SYSTEM ASM_MVCDR (* Assembly System Control+Diagnostics+HMI with Remote Model+View *)
  (* Standard: 61499-1; Classification: Simulation; ApplicationDomain: Assembly; Type: Dual Stroke Cylinder *)
  (* Version 0.1, 2004-10-21, JHC, Rockwell Automation, Adapted to new Load/Unload model. *)
  (* Version 0.0, 2004-09-26, JHC, Rockwell Automation, Extended from ASM_MVCDL1. *)
  DEVICE DIAGNOSTICS : FRAME_DEVICE
    RESOURCE IO : EMB_RES
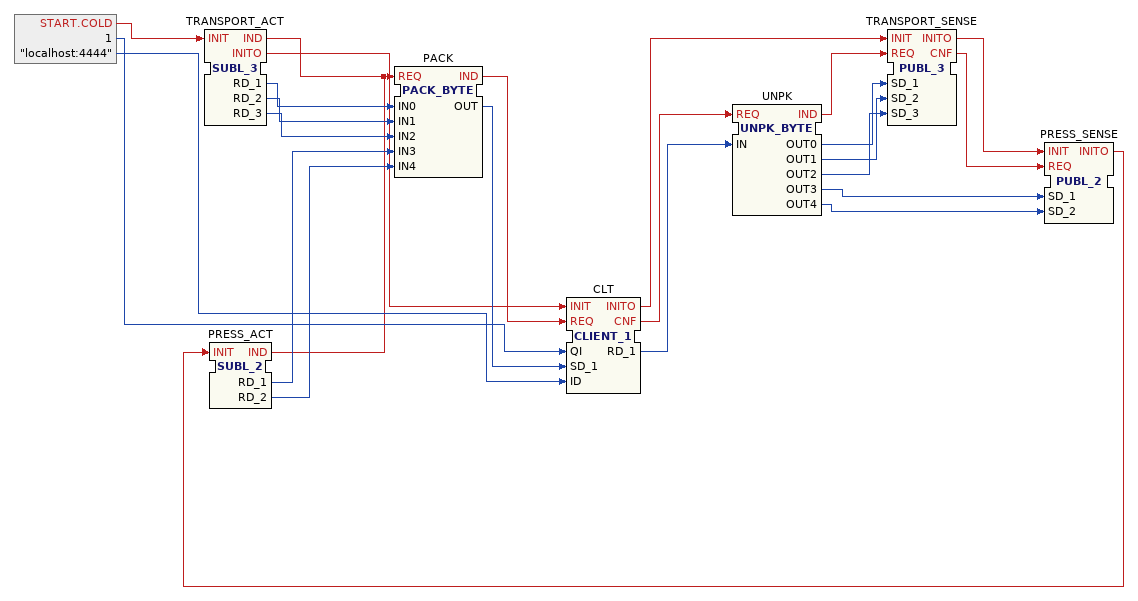
      FBS
        TRANSPORT_SENSE : PUBL_3;
        TRANSPORT_ACT : SUBL_3;
        PRESS_ACT : SUBL_2;
        PRESS_SENSE : PUBL_2;
        PACK : PACK_BYTE;
        CLT : CLIENT_1;
        UNPK : UNPK_BYTE;
      END_FBS
      EVENT_CONNECTIONS
        START.COLD TO TRANSPORT_ACT.INIT;
        TRANSPORT_ACT.IND TO PACK.REQ;
        PRESS_ACT.IND TO PACK.REQ;
        TRANSPORT_ACT.INITO TO CLT.INIT;
        PACK.IND TO CLT.REQ;
        CLT.INITO TO TRANSPORT_SENSE.INIT;
        CLT.CNF TO UNPK.REQ;
        UNPK.IND TO TRANSPORT_SENSE.REQ;
        TRANSPORT_SENSE.INITO TO PRESS_SENSE.INIT;
        TRANSPORT_SENSE.CNF TO PRESS_SENSE.REQ;
        PRESS_SENSE.INITO TO PRESS_ACT.INIT;
      END_CONNECTIONS
      DATA_CONNECTIONS
        TRANSPORT_ACT.RD_1 TO PACK.IN0;
        TRANSPORT_ACT.RD_2 TO PACK.IN1;
        TRANSPORT_ACT.RD_3 TO PACK.IN2;
        PRESS_ACT.RD_1 TO PACK.IN3;
        PRESS_ACT.RD_2 TO PACK.IN4;
        1 TO CLT.QI;
        CLT.RD_1 TO UNPK.IN;
        UNPK.OUT0 TO TRANSPORT_SENSE.SD_1;
        UNPK.OUT1 TO TRANSPORT_SENSE.SD_2;
        UNPK.OUT2 TO TRANSPORT_SENSE.SD_3;
        UNPK.OUT3 TO PRESS_SENSE.SD_1;
        UNPK.OUT4 TO PRESS_SENSE.SD_2;
        PACK.OUT TO CLT.SD_1;
        "localhost:4444" TO CLT.ID;
      END_CONNECTIONS
    END_RESOURCE
    RESOURCE LOG : PANEL_RESOURCE
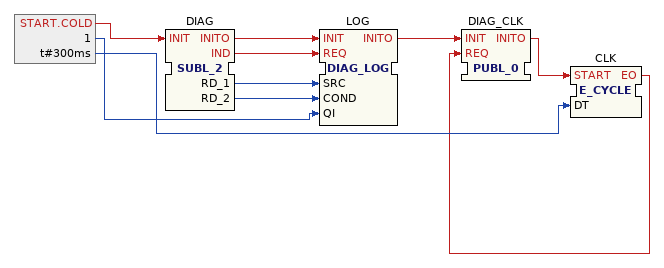
      FBS
        DIAG : SUBL_2;
        LOG : DIAG_LOG;
        CLK : E_CYCLE;
        DIAG_CLK : PUBL_0;
      END_FBS
      EVENT_CONNECTIONS
        START.COLD TO DIAG.INIT;
        DIAG.INITO TO LOG.INIT;
        DIAG.IND TO LOG.REQ;
        LOG.INITO TO DIAG_CLK.INIT;
        DIAG_CLK.INITO TO CLK.START;
        CLK.EO TO DIAG_CLK.REQ;
      END_CONNECTIONS
      DATA_CONNECTIONS
        DIAG.RD_1 TO LOG.SRC;
        DIAG.RD_2 TO LOG.COND;
        1 TO LOG.QI;
        t#300ms TO CLK.DT; (* Stretched 20% from MODEL.CLOCK.CLK.DT *)
      END_CONNECTIONS
    END_RESOURCE
    RESOURCE MONITOR : EMB_RES
      FBS
        PRESS : MECH2_DIAGL;
        TRANSPORT : DSCYL_DIAGL;
      END_FBS
      EVENT_CONNECTIONS
        START.COLD TO PRESS.INIT;
        PRESS.INITO TO TRANSPORT.INIT;
      END_CONNECTIONS
      DATA_CONNECTIONS
        "DIAG" TO PRESS.DIAG_ID;
        "PRESS" TO PRESS.SRC;
        "DIAG" TO TRANSPORT.DIAG_ID;
        "TRANSPORT" TO TRANSPORT.SRC;
        10 TO PRESS.NF;
        10 TO PRESS.NR;
        10 TO TRANSPORT.NF1;
        10 TO TRANSPORT.NF2;
        10 TO TRANSPORT.NR;
      END_CONNECTIONS
    END_RESOURCE
    DATA_CONNECTIONS
      1 TO LOG.ROWS;
      1 TO LOG.COLS;
    END_CONNECTIONS
  END_DEVICE
  DEVICE CONTROL : FRAME_DEVICE
    RESOURCE ASSY_CTL : EMB_RES
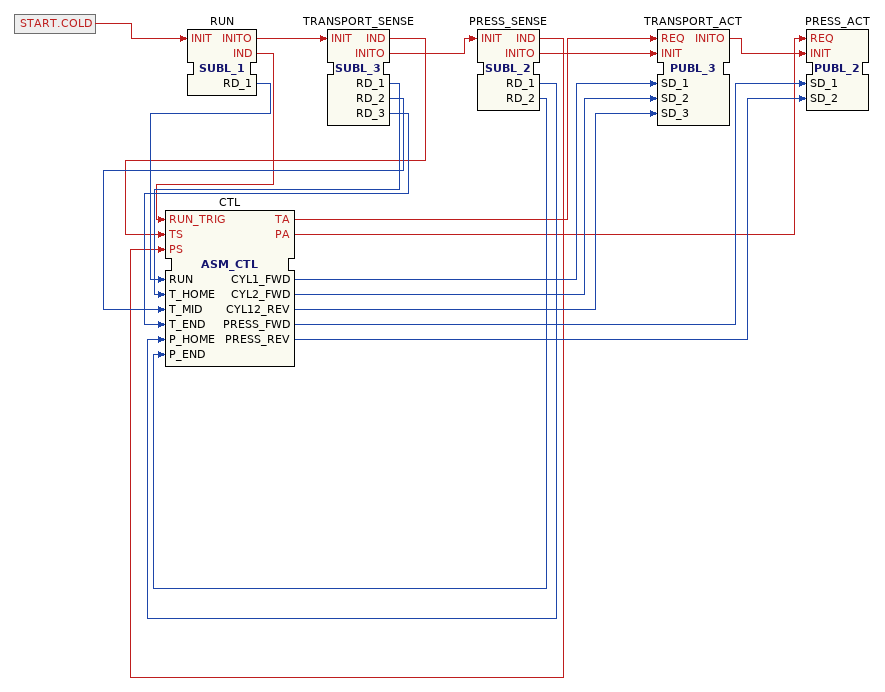
      FBS
        TRANSPORT_SENSE : SUBL_3;
        PRESS_SENSE : SUBL_2;
        TRANSPORT_ACT : PUBL_3;
        PRESS_ACT : PUBL_2;
        CTL : ASM_CTL;
        RUN : SUBL_1;
      END_FBS
      EVENT_CONNECTIONS
        TRANSPORT_SENSE.IND TO CTL.TS;
        CTL.TA TO TRANSPORT_ACT.REQ;
        CTL.PA TO PRESS_ACT.REQ;
        START.COLD TO RUN.INIT;
        RUN.INITO TO TRANSPORT_SENSE.INIT;
        RUN.IND TO CTL.RUN_TRIG;
        TRANSPORT_SENSE.INITO TO PRESS_SENSE.INIT;
        PRESS_SENSE.IND TO CTL.PS;
        PRESS_SENSE.INITO TO TRANSPORT_ACT.INIT;
        TRANSPORT_ACT.INITO TO PRESS_ACT.INIT;
      END_CONNECTIONS
      DATA_CONNECTIONS
        CTL.CYL1_FWD TO TRANSPORT_ACT.SD_1;
        CTL.CYL2_FWD TO TRANSPORT_ACT.SD_2;
        CTL.CYL12_REV TO TRANSPORT_ACT.SD_3;
        CTL.PRESS_FWD TO PRESS_ACT.SD_1;
        CTL.PRESS_REV TO PRESS_ACT.SD_2;
        TRANSPORT_SENSE.RD_1 TO CTL.T_HOME;
        TRANSPORT_SENSE.RD_2 TO CTL.T_MID;
        TRANSPORT_SENSE.RD_3 TO CTL.T_END;
        PRESS_SENSE.RD_1 TO CTL.P_HOME;
        PRESS_SENSE.RD_2 TO CTL.P_END;
        RUN.RD_1 TO CTL.RUN;
      END_CONNECTIONS
    END_RESOURCE
    RESOURCE TRANSPORT_SENSORS : PANEL_RESOURCE
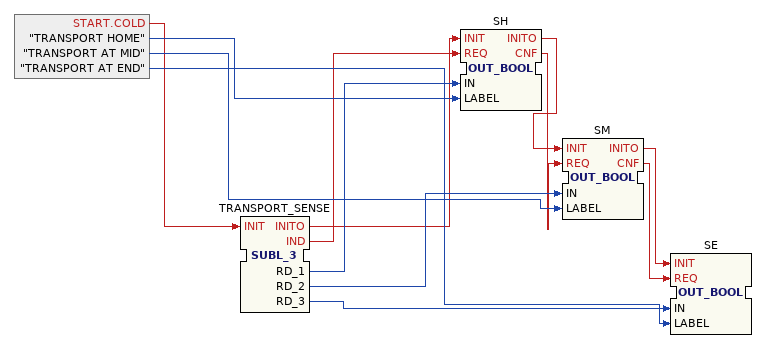
      FBS
        TRANSPORT_SENSE : SUBL_3;
        SH : OUT_BOOL;
        SM : OUT_BOOL;
        SE : OUT_BOOL;
      END_FBS
      EVENT_CONNECTIONS
        START.COLD TO TRANSPORT_SENSE.INIT;
        TRANSPORT_SENSE.INITO TO SH.INIT;
        SH.INITO TO SM.INIT;
        SM.INITO TO SE.INIT;
        TRANSPORT_SENSE.IND TO SH.REQ;
        SH.CNF TO SM.REQ;
        SM.CNF TO SE.REQ;
      END_CONNECTIONS
      DATA_CONNECTIONS
        TRANSPORT_SENSE.RD_1 TO SH.IN;
        TRANSPORT_SENSE.RD_2 TO SM.IN;
        TRANSPORT_SENSE.RD_3 TO SE.IN;
        "TRANSPORT HOME" TO SH.LABEL;
        "TRANSPORT AT MID" TO SM.LABEL;
        "TRANSPORT AT END" TO SE.LABEL;
      END_CONNECTIONS
    END_RESOURCE
    RESOURCE TRANSPORT_ACTUATORS : PANEL_RESOURCE
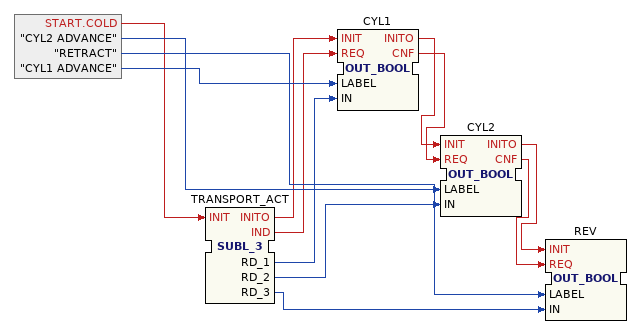
      FBS
        CYL1 : OUT_BOOL;
        CYL2 : OUT_BOOL;
        REV : OUT_BOOL;
        TRANSPORT_ACT : SUBL_3;
      END_FBS
      EVENT_CONNECTIONS
        CYL1.INITO TO CYL2.INIT;
        CYL2.INITO TO REV.INIT;
        CYL2.CNF TO REV.REQ;
        CYL1.CNF TO CYL2.REQ;
        START.COLD TO TRANSPORT_ACT.INIT;
        TRANSPORT_ACT.INITO TO CYL1.INIT;
        TRANSPORT_ACT.IND TO CYL1.REQ;
      END_CONNECTIONS
      DATA_CONNECTIONS
        "CYL2 ADVANCE" TO CYL2.LABEL;
        "RETRACT" TO REV.LABEL;
        "CYL1 ADVANCE" TO CYL1.LABEL;
        TRANSPORT_ACT.RD_1 TO CYL1.IN;
        TRANSPORT_ACT.RD_2 TO CYL2.IN;
        TRANSPORT_ACT.RD_3 TO REV.IN;
      END_CONNECTIONS
    END_RESOURCE
    RESOURCE PRESS_SENSORS : PANEL_RESOURCE
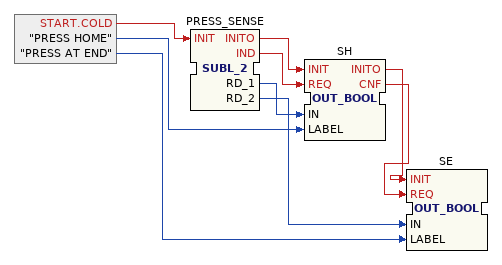
      FBS
        PRESS_SENSE : SUBL_2;
        SH : OUT_BOOL;
        SE : OUT_BOOL;
      END_FBS
      EVENT_CONNECTIONS
        START.COLD TO PRESS_SENSE.INIT;
        PRESS_SENSE.INITO TO SH.INIT;
        SH.INITO TO SE.INIT;
        PRESS_SENSE.IND TO SH.REQ;
        SH.CNF TO SE.REQ;
      END_CONNECTIONS
      DATA_CONNECTIONS
        PRESS_SENSE.RD_1 TO SH.IN;
        PRESS_SENSE.RD_2 TO SE.IN;
        "PRESS HOME" TO SH.LABEL;
        "PRESS AT END" TO SE.LABEL;
      END_CONNECTIONS
    END_RESOURCE
    RESOURCE PRESS_ACTUATORS : PANEL_RESOURCE
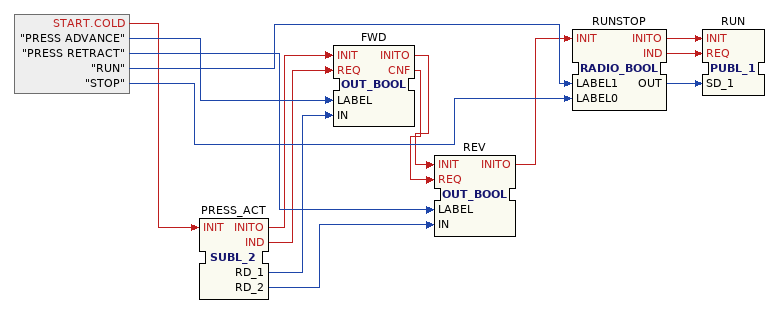
      FBS
        FWD : OUT_BOOL;
        REV : OUT_BOOL;
        PRESS_ACT : SUBL_2;
        RUNSTOP : RADIO_BOOL;
        RUN : PUBL_1;
      END_FBS
      EVENT_CONNECTIONS
        FWD.INITO TO REV.INIT;
        FWD.CNF TO REV.REQ;
        START.COLD TO PRESS_ACT.INIT;
        PRESS_ACT.INITO TO FWD.INIT;
        PRESS_ACT.IND TO FWD.REQ;
        REV.INITO TO RUNSTOP.INIT;
        RUNSTOP.INITO TO RUN.INIT;
        RUNSTOP.IND TO RUN.REQ;
      END_CONNECTIONS
      DATA_CONNECTIONS
        "PRESS ADVANCE" TO FWD.LABEL;
        "PRESS RETRACT" TO REV.LABEL;
        PRESS_ACT.RD_1 TO FWD.IN;
        PRESS_ACT.RD_2 TO REV.IN;
        "RUN" TO RUNSTOP.LABEL1;
        "STOP" TO RUNSTOP.LABEL0;
        RUNSTOP.OUT TO RUN.SD_1;
      END_CONNECTIONS
    END_RESOURCE
    DATA_CONNECTIONS
      3 TO TRANSPORT_SENSORS.ROWS;
      1 TO TRANSPORT_SENSORS.COLS;
      3 TO TRANSPORT_ACTUATORS.ROWS;
      1 TO TRANSPORT_ACTUATORS.COLS;
    END_CONNECTIONS
  END_DEVICE
  DEVICE MODEL : RMT_FRAME
    RESOURCE IO : EMB_RES
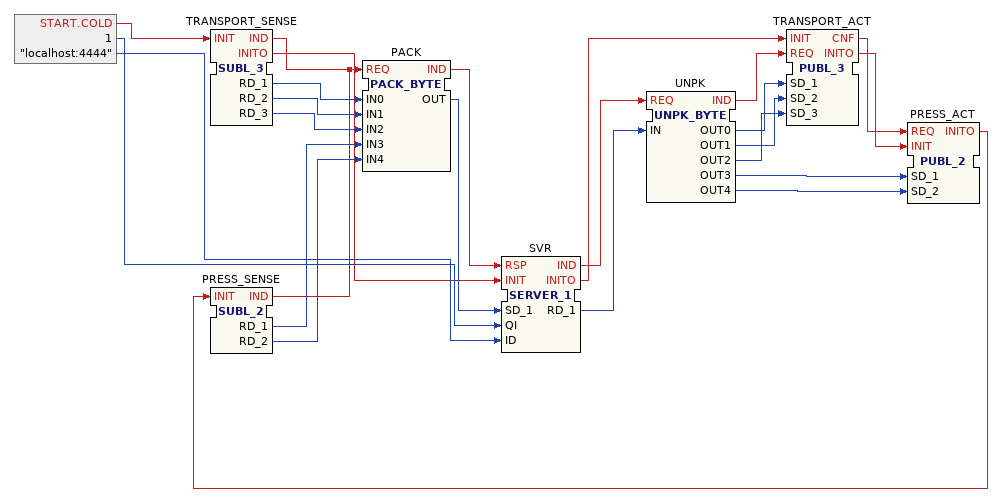
      FBS
        TRANSPORT_SENSE : SUBL_3;
        TRANSPORT_ACT : PUBL_3;
        PRESS_SENSE : SUBL_2;
        PRESS_ACT : PUBL_2;
        PACK : PACK_BYTE;
        SVR : SERVER_1;
        UNPK : UNPK_BYTE;
      END_FBS
      EVENT_CONNECTIONS
        START.COLD TO TRANSPORT_SENSE.INIT;
        TRANSPORT_SENSE.IND TO PACK.REQ;
        PRESS_SENSE.IND TO PACK.REQ;
        PACK.IND TO SVR.RSP;
        TRANSPORT_SENSE.INITO TO SVR.INIT;
        SVR.IND TO UNPK.REQ;
        SVR.INITO TO TRANSPORT_ACT.INIT;
        UNPK.IND TO TRANSPORT_ACT.REQ;
        TRANSPORT_ACT.CNF TO PRESS_ACT.REQ;
        TRANSPORT_ACT.INITO TO PRESS_ACT.INIT;
        PRESS_ACT.INITO TO PRESS_SENSE.INIT;
      END_CONNECTIONS
      DATA_CONNECTIONS
        TRANSPORT_SENSE.RD_1 TO PACK.IN0;
        TRANSPORT_SENSE.RD_2 TO PACK.IN1;
        TRANSPORT_SENSE.RD_3 TO PACK.IN2;
        PRESS_SENSE.RD_1 TO PACK.IN3;
        PRESS_SENSE.RD_2 TO PACK.IN4;
        PACK.OUT TO SVR.SD_1;
        1 TO SVR.QI;
        "localhost:4444" TO SVR.ID;
        SVR.RD_1 TO UNPK.IN;
        UNPK.OUT0 TO TRANSPORT_ACT.SD_1;
        UNPK.OUT1 TO TRANSPORT_ACT.SD_2;
        UNPK.OUT2 TO TRANSPORT_ACT.SD_3;
        UNPK.OUT3 TO PRESS_ACT.SD_1;
        UNPK.OUT4 TO PRESS_ACT.SD_2;
      END_CONNECTIONS
    END_RESOURCE
    RESOURCE CLOCK : EMB_RES
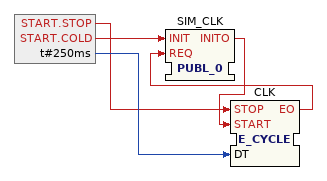
      FBS
        CLK : E_CYCLE;
        SIM_CLK : PUBL_0;
      END_FBS
      EVENT_CONNECTIONS
        START.STOP TO CLK.STOP;
        START.COLD TO SIM_CLK.INIT;
        SIM_CLK.INITO TO CLK.START;
        CLK.EO TO SIM_CLK.REQ;
      END_CONNECTIONS
      DATA_CONNECTIONS
        t#250ms TO CLK.DT;
      END_CONNECTIONS
    END_RESOURCE
    RESOURCE TRANSPORT_MDL : PANEL_RESOURCE
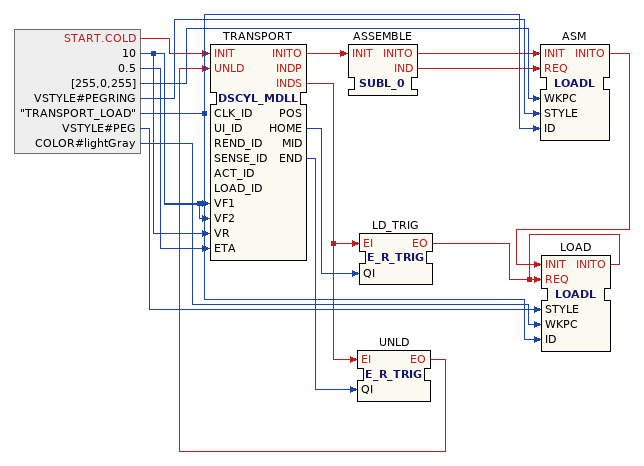
      FBS
        TRANSPORT : DSCYL_MDLL;
        UNLD : E_R_TRIG;
        ASM : LOADL;
        LD_TRIG : E_R_TRIG;
        ASSEMBLE : SUBL_0;
        LOAD : LOADL;
      END_FBS
      EVENT_CONNECTIONS
        TRANSPORT.INDS TO UNLD.EI;
        TRANSPORT.INDS TO LD_TRIG.EI;
        START.COLD TO TRANSPORT.INIT;
        TRANSPORT.INITO TO ASSEMBLE.INIT;
        ASSEMBLE.INITO TO ASM.INIT;
        ASSEMBLE.IND TO ASM.REQ;
        UNLD.EO TO TRANSPORT.UNLD;
        ASM.INITO TO LOAD.INIT;
        LOAD.INITO TO LOAD.REQ;
        LD_TRIG.EO TO LOAD.REQ;
      END_CONNECTIONS
      DATA_CONNECTIONS
        TRANSPORT.END TO UNLD.QI;
        TRANSPORT.HOME TO LD_TRIG.QI;
        10 TO TRANSPORT.VF1;
        10 TO TRANSPORT.VF2;
        10 TO TRANSPORT.VR;
        0.5 TO TRANSPORT.ETA;
        [255,0,255] TO ASM.WKPC;
        VSTYLE#PEGRING TO ASM.STYLE;
        "TRANSPORT_LOAD" TO ASM.ID;
        VSTYLE#PEG TO LOAD.STYLE;
        COLOR#lightGray TO LOAD.WKPC;
        "TRANSPORT_LOAD" TO LOAD.ID;
      END_CONNECTIONS
    END_RESOURCE
    RESOURCE PRESS_MDL : PANEL_RESOURCE
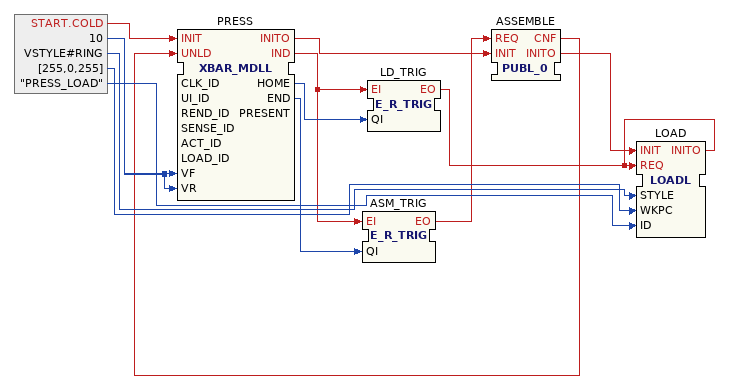
      FBS
        PRESS : XBAR_MDLL;
        ASM_TRIG : E_R_TRIG; (* Gate for assembly event *)
        ASSEMBLE : PUBL_0;
        LD_TRIG : E_R_TRIG;
        LOAD : LOADL;
      END_FBS
      EVENT_CONNECTIONS
        ASM_TRIG.EO TO ASSEMBLE.REQ;
        START.COLD TO PRESS.INIT;
        PRESS.IND TO LD_TRIG.EI;
        PRESS.IND TO ASM_TRIG.EI;
        PRESS.INITO TO ASSEMBLE.INIT;
        ASSEMBLE.CNF TO PRESS.UNLD;
        ASSEMBLE.INITO TO LOAD.INIT;
        LD_TRIG.EO TO LOAD.REQ;
        LOAD.INITO TO LOAD.REQ;
      END_CONNECTIONS
      DATA_CONNECTIONS
        PRESS.END TO ASM_TRIG.QI;
        10 TO PRESS.VF;
        10 TO PRESS.VR;
        PRESS.HOME TO LD_TRIG.QI;
        VSTYLE#RING TO LOAD.STYLE;
        [255,0,255] TO LOAD.WKPC;
        "PRESS_LOAD" TO LOAD.ID;
      END_CONNECTIONS
    END_RESOURCE
    RESOURCE ASSEMBLY : VIEW_PANEL
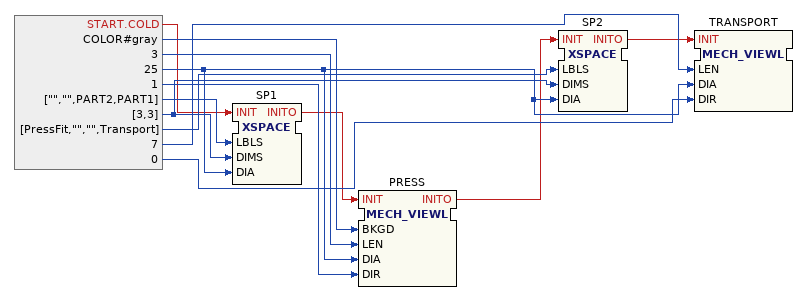
      FBS
        SP1 : XSPACE;
        PRESS : MECH_VIEWL; (* Vertical press element *)
        SP2 : XSPACE;
        TRANSPORT : MECH_VIEWL; (* Dual-Cylinder Transport Mechanism *)
      END_FBS
      EVENT_CONNECTIONS
        START.COLD TO SP1.INIT;
        SP1.INITO TO PRESS.INIT;
        PRESS.INITO TO SP2.INIT;
        SP2.INITO TO TRANSPORT.INIT;
      END_CONNECTIONS
      DATA_CONNECTIONS
        COLOR#gray TO PRESS.BKGD;
        3 TO PRESS.LEN;
        25 TO PRESS.DIA;
        1 TO PRESS.DIR;
        ["","",PART2,PART1] TO SP1.LBLS;
        [3,3] TO SP1.DIMS;
        25 TO SP1.DIA;
        [PressFit,"","",Transport] TO SP2.LBLS;
        [3,3] TO SP2.DIMS;
        25 TO SP2.DIA;
        7 TO TRANSPORT.LEN;
        25 TO TRANSPORT.DIA;
        0 TO TRANSPORT.DIR;
      END_CONNECTIONS
    END_RESOURCE
    DATA_CONNECTIONS
      0 TO ASSEMBLY.TRACE;
      25 TO ASSEMBLY.DIA;
      [7,5] TO ASSEMBLY.SIZE;
      0 TO ASSEMBLY.VERTICAL;
    END_CONNECTIONS
  END_DEVICE
  DATA_CONNECTIONS (* parameter values *)
    [380,100,185,150] TO MODEL.BOUNDS;
    [100,100,280,150] TO CONTROL.BOUNDS;
    [2,2] TO CONTROL.GRID;
    [100,250,465,150] TO DIAGNOSTICS.BOUNDS;
    [1,1] TO DIAGNOSTICS.GRID;
  END_CONNECTIONS
END_SYSTEM
